TYPE DatabaseThroughput EXTENDS DataTag:
STRUCT
	{attribute 'FieldName' := 'DB_queue_count'}
    db_insert_queue_count: UDINT;
	{attribute 'FieldName' := 'DB_buffer_current_index'}
    current_index: UDINT;
	{attribute 'FieldName' := 'DB_buffer_next_index'}
    next_index: UDINT;
END_STRUCT
END_TYPE

(* stored: Version 1.1.0.1, ProductVersion 3.1.4024.12
   DUT DatabaseThroughput: Id {39ced11c-3b33-4086-a1c0-e6d1ba5f33fd} *)
